ABB RobotStudio station: FigurDrawV7.5CodeDone.rsstn

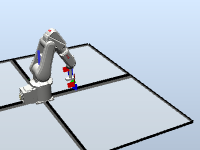
Station Ny63 (saved by RobotStudio 6.8.8307.1040)
Controller 120-100761
  mechanical unit ROB_1: IRB120_3_58__01, 6 joints, base frame (0, 0, 0) mm
Layout (positions relative to the parent item):
  - IRB120_3_58__01 [mechanism, from Robots\IRB120_3_58_G_01.rslib] at (0, 0, 0) mm; joint values [0, 0.3343, 0.705, 0, 0.5315, 0] (rad or m)
  - Tusch3 [mechanism, from Libraries\Tusch3.rslib] at (302, 0, 248.2) mm, rotated rx 180 ry 0 rz 180 deg
Attachment: Tusch3 is attached to IRB120_3_58__01 / Link6
Targets, tools, work objects and paths stored in the station, written as RAPID:
! task T_ROB1
MODULE MainModule
  PROC main()
  ENDPROC
ENDMODULE

! task T_ROB1
MODULE CalibData
  PERS tooldata Tusch3:=[TRUE,[[-40.7,0,181.64],[1,0,0,0]],[0.6,[14,0,78.3],[1,0,0,0],0.007,0.01,0.01]];
ENDMODULE

